TYPE ST_OEE :
STRUCT
	dtLastReset: DATE_AND_TIME;
	nNumCycles: UDINT;
	nHrsAvailable: REAL;
	nHrsUtilised: REAL;
	nHrsFaulted: REAL;
END_STRUCT
END_TYPE

(* stored: Version 1.1.0.1, ProductVersion 3.1.4024.12
   DUT ST_OEE: Id {dacef7f6-bf2c-4124-a48e-df1d1b2384f7} *)
